# EPICS autosave request: ipApp/Db/KeyenceCL3000_chan_settings.req
$(P)$(S):$(CHAN):measurement.SCAN
$(P)$(S):$(CHAN):measType
$(P)$(S):$(CHAN):offset_set
$(P)$(S):$(CHAN):scaling_set
